Fanuc KAREL source: kt00741.KL

-- PROVISIONAL review KL for V1013-1; original PC SHA256 8c99360abc3f1f2df624c92399a2b77bd2ba0d77019cf80ab0165ff5c2aacc12
-- Incomplete behavior may be omitted. Consult companion uncertainty JSON. Do not deploy.
PROGRAM KT00741
%NOLOCKGROUP
VAR
  OUT : INTEGER
-- UNRESOLVED_DECL ARG type=002017
BEGIN
  -- UNRESOLVED_PC offsets 5-18; opcodes 22,1D,23
  -- UNRESOLVED_PC offsets 23-27; opcodes 7F
END KT00741
